{attribute 'hide_all_locals'}
FUNCTION_BLOCK FB_1_COMM EXTENDS FB_0_BASE 
// IMPLEMENTS ITF_1_Communication

VAR_INPUT
	SET_C: stSettings_Comm;
    DEBUG_COMM : DEBUG_COMM;

END_VAR


VAR_OUTPUT
	{attribute 'OPC.UA.DA' := '1'}
	HMI_COMM: stHMI_COMM;
END_VAR
VAR
    // Desired state from Robot / lifecycle
    _ConnectionRequested : BOOL;

    // Request sent toward the child communication implementation
    bRequestConnection : BOOL;

    // Feedback supplied by the child communication implementation
    

    // Reconnect sequencing
    _ReconnectRequested : BOOL;

    // Communication state
    _eCommState : E_CommState := E_CommState.eDisconnected;
	// Transient communication faults recover automatically. After the configured
    // number of failed reconnect attempts the fault escalates to ErrorProcessing
    // and requires an operator Reset/Acknowledge.
    _nAutoReconnectAttempts : UINT;
	
    // Timers
    _tonConnectTimeout    : TON;
    _tonDisconnectTimeout : TON;
    _tonReconnectDelay    : TON;
    _tonStopTimeout       : TON;

    

    // Generic command transport lifecycle. Concrete COMM adapters update these fields.
    // IDs/results remain latched until the next command is locally accepted.
    _commCanAcceptCommand   : BOOL := TRUE;
    _commAcceptedCommandID  : UINT;
    _commActiveCommandID    : UINT;
    _commCommandBusy        : BOOL;
    _commCommandState       : eProgress := INIT;
    _commCommandResult      : eResult := NONE;

    // Functional stop lifecycle. A software stop is never safety-rated.
    _stopPending            : BOOL;
    _stopMode               : eStopMode := eStopMode.ControlledStop;
    _stopCommandID          : UINT;
    _stopStarted            : BOOL;
    _stopFailed             : BOOL;
    _motionStopped          : BOOL := TRUE;
	_bConnected: BOOL;
	_Init_Comm: BOOL;
END_VAR

PROPERTY AcceptedCommandID : UINT
GET
AcceptedCommandID := _commAcceptedCommandID;
END_GET
SET
_commAcceptedCommandID := AcceptedCommandID;
END_SET
END_PROPERTY

PROPERTY ActiveCommandID : UINT
GET
ActiveCommandID := _commActiveCommandID;
END_GET
SET
 _commActiveCommandID:=ActiveCommandID;
END_SET
END_PROPERTY

PROPERTY Busy : BOOL
GET
Busy :=
    _commCommandBusy
    OR _stopPending
    OR (_eCommState = E_CommState.eConnecting)
    OR (_eCommState = E_CommState.eDisconnecting)
    OR (_eCommState = E_CommState.eReconnectWait);
END_GET
SET
_commCommandBusy := Busy;
IF Busy AND NOT _stopPending THEN
    _motionStopped := FALSE;
END_IF
END_SET
END_PROPERTY

PROPERTY CanAcceptCommand : BOOL
GET
CanAcceptCommand :=
            Operational
            AND _commCanAcceptCommand
            AND NOT Busy
            AND NOT _stopPending;
END_GET
SET
_commCanAcceptCommand := CanAcceptCommand;
END_SET
END_PROPERTY

PROPERTY CommandResult : eResult
GET
CommandResult := _commCommandResult;
END_GET
SET
 _commCommandResult := CommandResult;
END_SET
END_PROPERTY

PROPERTY CommandState : eProgress
GET
CommandState := _commCommandState;
END_GET
SET
_commCommandState := CommandState;
END_SET
END_PROPERTY

METHOD Connect : BOOL

_ConnectionRequested := TRUE;

Connect := TRUE;
END_METHOD

PROPERTY Connected : BOOL
GET
IF DEBUG_COMM.bSimConnected THEN
    Connected := _ConnectionRequested;
ELSE
    Connected := _bConnected;
END_IF
END_GET
SET
_bConnected := Connected;
END_SET
END_PROPERTY

ACTION CYCLIC_COMM:
IF NOT _Init_Comm THEN
	_Init_Comm:=TRUE;
	SETUP_COMM();
END_IF

CYCLIC_BASE();


// --------------------------------------------------
// Timers
// --------------------------------------------------

_tonConnectTimeout(
    IN := _eCommState = E_CommState.eConnecting,
    PT := SET_C.tConnectTimeout
	
);

_tonDisconnectTimeout(
    IN := _eCommState = E_CommState.eDisconnecting,
    PT := SET_C.tDisconnectTimeout
);

_tonReconnectDelay(
    IN := _eCommState = E_CommState.eReconnectWait,
    PT := SET_C.tReconnectDelay
);

_tonStopTimeout(
    IN := _stopPending AND _stopStarted AND NOT _stopFailed,
    PT := SET_C.tStopTimeout
);

// Complete the stop through the concrete communication adapter.
IF _stopPending THEN
    _stopFailed := HasPhysicalStopFailed() OR _tonStopTimeout.Q;

    IF _stopFailed THEN
        IF _tonStopTimeout.Q THEN
            Messenger.AddError(eMessageCategories.TimeoutFailure, CONCAT(Path, '.StopMotion'),
                'Physical stop timed out');
        ELSE
            Messenger.AddError(eMessageCategories.HardwareFailure, CONCAT(Path, '.StopMotion'),
                'Physical stop failed');
        END_IF

        IF _stopCommandID <> 0 THEN
            CommandState := eProgress.FINALIZED;
            CommandResult := eResult.ERROR;
            ActiveCommandID := 0;
        END_IF
        _commCommandBusy := FALSE;
        _stopPending := FALSE;

    ELSIF IsPhysicalStopComplete() THEN
        _motionStopped := TRUE;
        IF _stopCommandID <> 0 THEN
            CommandState := eProgress.ABORTED;
            CommandResult := eResult.FAILURE;
            ActiveCommandID := 0;
        END_IF
        _commCommandBusy := FALSE;
        _stopPending := FALSE;
    END_IF
END_IF





// --------------------------------------------------
// Communication state machine
// --------------------------------------------------

CASE _eCommState OF


    // ==============================================
    // DISCONNECTED
    // ==============================================
    E_CommState.eDisconnected:

        bRequestConnection := FALSE;

        IF _ReconnectRequested
           AND _ConnectionRequested THEN

            _eCommState := E_CommState.eReconnectWait;

        ELSIF _ConnectionRequested THEN

            bRequestConnection := TRUE;
            _eCommState := E_CommState.eConnecting;

        END_IF


    // ==============================================
    // CONNECTING
    // ==============================================
    E_CommState.eConnecting:

        bRequestConnection := TRUE;


        // User cancelled connection request
        IF NOT _ConnectionRequested THEN

            bRequestConnection := FALSE;
            _eCommState := E_CommState.eDisconnecting;


        // Communication fully initialized
        ELSIF Operational THEN

            // Link healthy again: clear any comm messages this component raised.
            _ReconnectRequested := FALSE;
            _nAutoReconnectAttempts := 0;
            _eCommState := E_CommState.eConnected;


        // Timeout
        ELSIF _tonConnectTimeout.Q THEN

            _nAutoReconnectAttempts := _nAutoReconnectAttempts + 1;
            bRequestConnection := FALSE;

            IF (SET_C.nMaxAutoReconnectAttempts > 0)
                AND (_nAutoReconnectAttempts >= SET_C.nMaxAutoReconnectAttempts) THEN

                // Automatic recovery is exhausted. Escalate once into ErrorProcessing;
                // the user must acknowledge before another configure/connect sequence.
                SetRecoveryMode(Mode := eRecoveryMode.AcknowledgeRequired);
                Messenger.AddError(eMessageCategories.TimeoutFailure, Name,
                    'Automatic communication recovery exhausted; operator reset required');
                _ReconnectRequested := FALSE;
                _ConnectionRequested := FALSE;
            ELSE
                Messenger.AddWarn(eMessageCategories.TimeoutFailure, Name,
                    'Connection attempt timed out, retrying automatically');

                IF _ConnectionRequested THEN
                    _ReconnectRequested := TRUE;
                END_IF
            END_IF

            _eCommState := E_CommState.eDisconnecting;

        END_IF


    // ==============================================
    // CONNECTED
    // ==============================================
    E_CommState.eConnected:

        bRequestConnection := TRUE;


        // Explicit reconnect
        IF _ReconnectRequested THEN

            bRequestConnection := FALSE;
            _eCommState := E_CommState.eDisconnecting;


        // Explicit disconnect
        ELSIF NOT _ConnectionRequested THEN

            bRequestConnection := FALSE;
            _eCommState := E_CommState.eDisconnecting;


        // Unexpected loss of communication
        ELSIF NOT HMI_COMM._CommunicationConnected THEN

            // A single runtime link loss is recoverable. Keep the lifecycle alive and
            // reconnect internally; repeated connect failures escalate through the timeout path.
            Messenger.AddWarn(eMessageCategories.LostConnection, Name,
                'Communication lost; automatic reconnect started');

            bRequestConnection := FALSE;
            _ReconnectRequested := TRUE;

            _eCommState := E_CommState.eDisconnecting;

        END_IF


    // ==============================================
    // DISCONNECTING
    // ==============================================
    E_CommState.eDisconnecting:

        bRequestConnection := FALSE;


        IF NOT HMI_COMM._CommunicationConnected THEN

            IF _ReconnectRequested
               AND _ConnectionRequested THEN

                _eCommState := E_CommState.eReconnectWait;

            ELSE

                _ReconnectRequested := FALSE;
                _eCommState := E_CommState.eDisconnected;

            END_IF


        ELSIF _tonDisconnectTimeout.Q THEN

            Messenger.AddWarn(eMessageCategories.TimeoutFailure, Name, 'Disconnect timed out');

            // Stay in Disconnecting.
            // Do NOT falsely report Disconnected.

        END_IF


    // ==============================================
    // RECONNECT DELAY
    // ==============================================
    E_CommState.eReconnectWait:

        bRequestConnection := FALSE;


        // Reconnect cancelled
        IF NOT _ConnectionRequested THEN

            _ReconnectRequested := FALSE;
            _eCommState := E_CommState.eDisconnected;


        // Delay complete
        ELSIF _tonReconnectDelay.Q THEN

            _ReconnectRequested := FALSE;

            bRequestConnection := TRUE;
            _eCommState := E_CommState.eConnecting;

        END_IF


END_CASE
END_ACTION

METHOD Disconnect : BOOL
_ConnectionRequested := FALSE;
_ReconnectRequested := FALSE;

Disconnect := TRUE;
END_METHOD

METHOD PROTECTED EnsurePhysicalStopForLifecycle : BOOL
EnsurePhysicalStopForLifecycle := FALSE;

IF MotionStopped THEN
    EnsurePhysicalStopForLifecycle := TRUE;
    RETURN;
END_IF

IF NOT StopPending AND NOT StopMotion() THEN
    Messenger.AddError(
        eMessageCategories.HardwareFailure,
        CONCAT(Path, '.StopMotion'),
        'Communication adapter rejected the lifecycle stop request');
    RETURN;
END_IF

EnsurePhysicalStopForLifecycle := MotionStopped;
END_METHOD

PROPERTY MotionStopped : BOOL
GET
MotionStopped := _motionStopped AND NOT _stopPending;
END_GET
END_PROPERTY

METHOD PROTECTED OnActivate : eResult
VAR_INPUT
END_VAR

VAR
	eParentResult: eResult;
	myResult: ERESULT;
END_VAR

VAR //YOUR CODE
	succ : BOOL;
END_VAR
eParentResult := SUPER^.OnActivate();
//--------------------------------------------------
myResult:=NONE;
// ----- YOUR CODE HERE (incl. Alarms) -------------


myResult:=SUCCESS;

// ----- END YOUR CODE -----------------------------
//--------------------------------------------------
OnActivate := CombineResults(eParentResult,myResult);
END_METHOD

METHOD PROTECTED OnCleanup : eResult
VAR_INPUT
END_VAR

VAR
	eParentResult: eResult;
	myResult: ERESULT;
END_VAR

VAR //YOUR CODE
	succ : BOOL;
END_VAR
eParentResult := SUPER^.OnCleanup();
//--------------------------------------------------
myResult:=NONE;
// ----- YOUR CODE HERE (incl. Alarms) -------------

Disconnect();
IF NOT Connected THEN
	myResult:=SUCCESS;
END_IF

// ----- END YOUR CODE -----------------------------
//--------------------------------------------------
OnCleanup := CombineResults(eParentResult,myResult);
END_METHOD

METHOD PROTECTED OnConfigure : eResult
VAR_INPUT
END_VAR

VAR
	eParentResult: eResult;
	myResult: ERESULT;
END_VAR

VAR //YOUR CODE
	succ : BOOL;
END_VAR
eParentResult := SUPER^.OnConfigure();
//--------------------------------------------------
myResult:=NONE;
// ----- YOUR CODE HERE (incl. Alarms) -------------

Connect();
IF Operational  THEN
	myResult:=SUCCESS;
END_IF


// ----- END YOUR CODE -----------------------------
//--------------------------------------------------
OnConfigure := CombineResults(eParentResult,myResult);
END_METHOD

METHOD PROTECTED OnDeactivate : eResult
VAR_INPUT
END_VAR

VAR
	eParentResult: eResult;
	myResult: ERESULT;
END_VAR

VAR //YOUR CODE
	succ : BOOL;
END_VAR
eParentResult := SUPER^.OnDeactivate();
//--------------------------------------------------
myResult:=NONE;
// ----- YOUR CODE HERE (incl. Alarms) -------------

IF EnsurePhysicalStopForLifecycle() THEN
  myResult:=SUCCESS;
END_IF

// ----- END YOUR CODE -----------------------------
//--------------------------------------------------
OnDeactivate := CombineResults(eParentResult,myResult);
END_METHOD

METHOD PROTECTED OnError : eResult
VAR_INPUT
END_VAR

VAR
	eParentResult: eResult;
	myResult: ERESULT;
END_VAR

VAR //YOUR CODE
	succ : BOOL;
END_VAR
eParentResult := SUPER^.OnError();
      myResult := NONE;

      IF NOT EnsurePhysicalStopForLifecycle() THEN
          OnError := CombineResults(eParentResult, myResult);
          RETURN;
      END_IF

// Generic communication recovery is always a controlled disconnect. Reconnect is
// performed later by Configure; OnError never resumes a previous robot command.
Disconnect();

IF NOT Connected THEN
    _ReconnectRequested := FALSE;
    _ConnectionRequested := FALSE;
    bRequestConnection := FALSE;
    _eCommState := E_CommState.eDisconnected;
    _nAutoReconnectAttempts := 0;
    myResult := SUCCESS;
END_IF

OnError := CombineResults(eParentResult, myResult);
END_METHOD

METHOD PROTECTED OnShutdown : eResult
VAR_INPUT
END_VAR

    VAR
    	eParentResult: eResult;
    	myResult: ERESULT;
    END_VAR

    VAR //YOUR CODE
    	succ : BOOL;
    END_VAR
eParentResult := SUPER^.OnShutdown();
    //--------------------------------------------------
    myResult:=NONE;
    // ----- YOUR CODE HERE (incl. Alarms) -------------

  IF NOT EnsurePhysicalStopForLifecycle() THEN
    OnShutdown := CombineResults(eParentResult, myResult);
    RETURN;
  END_IF

Disconnect();
IF NOT Connected THEN
	myResult:=SUCCESS;
END_IF

// ----- END YOUR CODE -----------------------------
//--------------------------------------------------
OnShutdown := CombineResults(eParentResult,myResult);
END_METHOD

PROPERTY Operational : BOOL
SET
SUPER^.Operational:= Operational AND Connected;
END_SET
END_PROPERTY

METHOD Reconnect : BOOL
_ConnectionRequested := TRUE;
_ReconnectRequested := TRUE;

Reconnect := TRUE;
END_METHOD

PROPERTY RequestConnection : BOOL
GET
RequestConnection := bRequestConnection;
END_GET
SET
 bRequestConnection := RequestConnection;
END_SET
END_PROPERTY

METHOD PUBLIC ResetCommunication : BOOL
// Never erase evidence of a stop that has not reached standstill.
      IF _stopPending THEN
          ResetCommunication := FALSE;
          RETURN;
      END_IF

      // Generic reset: discard transport-command bookkeeping and request a clean reconnect.
// This does NOT reset robot/controller safety conditions.
CanAcceptCommand := TRUE;
AcceptedCommandID := 0;
ActiveCommandID := 0;

CommandState := INIT;
CommandResult := NONE;
Reconnect();
ResetCommunication := TRUE;
END_METHOD

PROPERTY SafetyStopActive : BOOL
GET
SafetyStopActive := ReadSafetyStopActive();
END_GET
END_PROPERTY

ACTION SETUP_COMM:

END_ACTION

METHOD PROTECTED StartPhysicalStop : BOOL
VAR_INPUT
    Mode : eStopMode;
END_VAR
StartPhysicalStop := TRUE;
END_METHOD

METHOD PROTECTED IsPhysicalStopComplete : BOOL
IsPhysicalStopComplete := TRUE;
END_METHOD

METHOD PROTECTED HasPhysicalStopFailed : BOOL
HasPhysicalStopFailed := FALSE;
END_METHOD

METHOD PROTECTED ReadSafetyStopActive : BOOL
ReadSafetyStopActive := FALSE;
END_METHOD

METHOD PUBLIC StopMotion : BOOL
StopMotion := FALSE;

IF _stopPending THEN
    StopMotion := TRUE;
    RETURN;
END_IF

IF NOT StartPhysicalStop(Mode := eStopMode.ControlledStop) THEN
    RETURN;
END_IF

_stopPending := TRUE;
_stopMode := eStopMode.ControlledStop;
_stopCommandID := ActiveCommandID;
_stopStarted := TRUE;
_stopFailed := FALSE;
_motionStopped := FALSE;

IF _stopCommandID <> 0 THEN
    CommandResult := eResult.NONE;
END_IF

_tonStopTimeout(IN := FALSE);
StopMotion := TRUE;
END_METHOD

PROPERTY StopPending : BOOL
GET
StopPending := _stopPending;
END_GET
END_PROPERTY

END_FUNCTION_BLOCK

(* stored: Version 1.1.0.1, ProductVersion 3.1.4026.18
   POU FB_1_COMM: Id {73f52913-3875-44cd-a06c-142e4cd90d86}, SpecialFunc None
   Folder FINAL: Id {d7990c19-4461-4ef9-a9c3-41dd59eb7d2b}
   Folder MotionControl: Id {9ebe1908-93ac-4cf6-a7d5-d0a567358124}
   Folder OVERRIDE: Id {e2759980-4448-4b35-8dbf-1dfc78f02aca}
   Folder StateControl: Id {c1b69548-4ff3-4256-aac8-59814ba2c761}
   Property AcceptedCommandID: Id {60d7e86d-2ef6-4d6f-bb21-251c22802799}
   Get Get: Id {8ce6a3a0-b19a-45ac-9d9d-9e72d8d8020c}
   Set Set: Id {258a74e7-c3d7-4278-be80-d424dc4b64e0}
   Property ActiveCommandID: Id {8c2c9e7e-d92a-463d-a9f9-5cb3ad54a055}
   Get Get: Id {99a81894-3218-4ebb-9c35-29038eb5479e}
   Set Set: Id {4a964539-a199-49d0-9456-608f00b9c1d0}
   Property Busy: Id {57cf1565-bfdf-43e0-b8be-60c84950548e}
   Get Get: Id {33a32cb5-dcf8-4f92-b164-a220f8b7b981}
   Set Set: Id {591498ad-c58c-4078-81de-4fbf8227f63f}
   Property CanAcceptCommand: Id {e36b9102-7992-44e5-8a2f-0ad461767e6c}
   Get Get: Id {3dd26639-26ba-43fe-a217-d9d0461e2052}
   Set Set: Id {bbffabb9-2c8c-4c46-a5d3-734cc365cf61}
   Property CommandResult: Id {ef906cf3-c3b7-4110-a2da-473905a396c7}
   Get Get: Id {460a019c-ad56-4214-8d20-9adaabd86832}
   Set Set: Id {d5f78c96-3d3f-4293-88f6-5dca2ac0ef57}
   Property CommandState: Id {e88b06bd-b100-4d6c-9b6e-88e9b6397a70}
   Get Get: Id {ebe78b68-751a-430d-9857-d1adb859ef46}
   Set Set: Id {6beb8faf-ee1a-4c5d-a238-db16292ed01a}
   Method Connect: Id {0e03e6e3-746a-4d15-b30d-e1d35cd9fa73}
   Property Connected: Id {12741b67-6a3c-4917-9eee-ef373e57c752}
   Get Get: Id {e2f59856-76f0-4d1d-a064-5db7172878ee}
   Set Set: Id {ecd2f951-5c05-47a3-ade8-e26970503204}
   Action CYCLIC_COMM: Id {2920dcfd-53c5-448d-9932-add88782955c}
   Method Disconnect: Id {3e0f527d-159a-4d89-8a65-81b0aeb4a5da}
   Method EnsurePhysicalStopForLifecycle: Id {b1124978-ea27-4b65-a747-64780794a32a}
   Property MotionStopped: Id {6f85e13b-3111-4868-89c6-48d06c5ec9cb}
   Get Get: Id {6b3f956f-c326-49b2-847a-f3f969004932}
   Method OnActivate: Id {4a1c3eeb-6c6d-4831-81db-3d184da3d943}
   Method OnCleanup: Id {ae58109b-b0e8-4811-8a5c-3770f3206063}
   Method OnConfigure: Id {a01179aa-e567-4321-93fd-631c3e2274ca}
   Method OnDeactivate: Id {6eb02c50-b291-4bcf-b1ad-138bb630e64a}
   Method OnError: Id {906994b9-e66f-4d00-8af4-b6fb49575473}
   Method OnShutdown: Id {5df962a8-b76a-42d4-b83d-c52e19cc1a66}
   Property Operational: Id {90ec2b27-bfaf-45b4-9aa5-21ddf3a8865d}
   Set Set: Id {4f19d267-1340-49ac-92ec-f176abd048d2}
   Method Reconnect: Id {1b214bc4-2670-4530-9e2e-4fb9a9440c51}
   Property RequestConnection: Id {f2ed25bd-6424-4266-a820-528a5d6767d6}
   Get Get: Id {3b6ef5bb-3136-4550-9ff2-b558ac527931}
   Set Set: Id {977d3991-b84d-40b2-bdff-5fcf47db105f}
   Method ResetCommunication: Id {ce234f47-9067-45ef-9d48-468fcefbc15a}
   Property SafetyStopActive: Id {5cc3821a-a232-4b40-a0f6-410fc5435fa2}
   Get Get: Id {4a028063-4176-4cb3-82ae-f7e0f0ca970e}
   Action SETUP_COMM: Id {8953db30-ebf8-4ae1-b477-95a9c5b6fb8c}
   Method StartPhysicalStop: Id {6d5b6f41-1418-4c48-bbc2-6114f0f7d8b1}
   Method IsPhysicalStopComplete: Id {71f60ec4-31d0-4e17-8b67-d728e2c25281}
   Method HasPhysicalStopFailed: Id {b5963943-a3ea-4c64-bb8c-83f43ac4a85d}
   Method ReadSafetyStopActive: Id {5059d265-c10c-4372-bf89-b2b839ae1ec7}
   Method StopMotion: Id {87fb0928-6cea-447d-8282-693d0d33345f}
   Property StopPending: Id {0d5ce5ca-c592-4ba5-acac-a6833088e4b8}
   Get Get: Id {53cd5606-782e-46bd-a25d-e4d09e237ba6} *)
